// TIA Portal V21 export
FUNCTION_BLOCK "PHT Block"   // FB401, LAD
{ S7_Optimized_Access := 'FALSE' }
// stored: AutoNumber false, SetENOAutomatically false
   VAR_INPUT
      Secs : Bool;
      Start : Bool;
      Stop : Bool;
      Abort : Bool;
      AlarmAck : Bool;
      AlwaysTrue : Bool;
      StartupMsgSelection : Bool;
      spare1 : Bool;
      spare2 : Bool;
      EndMsgSelection : Bool;
      EndMsgAck : Bool;
      Fault : Bool;
      Popup1Enable : Bool;
      Popup2Enable : Bool;
      ScadaHmi : Bool := 1;   // 0- scada, 1 - hmi
      StabilizeTime : Int;
      SetPressure : Real;
      ReleasePressure : Real;
      FailPressure : Real;
      AcceptableLeakage : Real;
      HoldTime : Int;
      UtilityValveDelay : Int;
      "Actual Minimum Pressure" : Real;
      "Actual Maximum Pressure" : Real;
      MaximumAttemptToFailedSelection : Int;
      MaximumNoAttemptToFailed : Int;
      PrintInterval : Int;
   END_VAR
   VAR_OUTPUT
      StartupMsg1 : Bool;
      CycleOver : Bool;
      LineValves : Bool;
      ControlValve : Bool;
      UtilityValve : Bool;
      StartupMsg : Bool;
      EndMsg : Bool;
      TestPassAlarm : Bool;
      TestFailAlarm : Bool;
      DrainValves : Bool;
      StartupMsg2 : Bool;
      StabilizeActualSecs : DInt;
      HoldActualMins : DInt;
      HoldActualSecs : DInt;
      Status : Int;
      StatusStr : String[60];
      UtilityValveActualDelay : Int;
      Event : Word;
   END_VAR
   VAR_IN_OUT
      Selected : Bool;
      CycleSelected : Bool;
      Running : Bool;
      VesselPressurised : Bool;
      DataLogCmd : Bool;
      StartLog : Bool;
      EndLog : Bool;
      DataLogYes : Bool;
      ResetPhtTimer : Bool;
      VesselStabilised : Bool;
      DelayToConfirmVesselPressurized : Bool;
      PressureDropDuringStabilizeTime : Bool;
      PressureDropDuringHoldTime : Bool;
      TestPassedRW : Bool;
      DelayToStartReleaseDone : Bool;
      DrainValve : Bool;
      StabilizePopup : Bool;
      LineValvesOpeningTime : Int;
      DrainValvesOpeningTime : Int;
      AcceptablePressure : Real;
      "PHT Selected" : Bool;
      TestAborted : Bool;
      ResetBit : Bool;
      Popup2Ack : Bool;
      StartupMsgYes : Bool;
      StartupMsgNo : Bool;
      MaximumNoAttemptToFailedTemp : Int;
   END_VAR
   VAR
      StabilizeTimer { S7_SetPoint := 'True'} : "R_TIMER";
      HoldTimer { S7_SetPoint := 'True'} : "R_TIMER";
      CheckPressureDuringStabilizeTime { S7_SetPoint := 'True'} : "On Delay Timer";
      CheckPressureDuringHoldTime { S7_SetPoint := 'True'} : "On Delay Timer";
      ReleaseCheckTime { S7_SetPoint := 'True'} : "On Delay Timer";
      CheckPressuredelay { S7_SetPoint := 'True'} : "On Delay Timer";
      DelayToStartRelease { S7_SetPoint := 'True'} : "On Delay Timer";
      StabilizeDelay { S7_SetPoint := 'True'} : "On Delay Timer";
      IEC_Timer_0_Instance { S7_SetPoint := 'True'} : TON_TIME;
      IEC_Timer_1_Instance { S7_SetPoint := 'True'} : TON_TIME;
      Timer1 { S7_SetPoint := 'True'} : TON_TIME;
      Timer2 { S7_SetPoint := 'True'} : TON_TIME;
      Timer3 { S7_SetPoint := 'True'} : TON_TIME;
      Timer4 { S7_SetPoint := 'True'} : TON_TIME;
      Timer5 { S7_SetPoint := 'True'} : TON_TIME;
      Timer6 { S7_SetPoint := 'True'} : TON_TIME;
      Timer7 { S7_SetPoint := 'True'} : TON_TIME;
      Re { ExternalAccessible := 'False'; ExternalVisible := 'False'; ExternalWritable := 'False'} : Bool;
      Re1 { ExternalAccessible := 'False'; ExternalVisible := 'False'; ExternalWritable := 'False'} : Bool;
      Re2 { ExternalAccessible := 'False'; ExternalVisible := 'False'; ExternalWritable := 'False'} : Bool;
      Re3 { ExternalAccessible := 'False'; ExternalVisible := 'False'; ExternalWritable := 'False'} : Bool;
      Re4 { ExternalAccessible := 'False'; ExternalVisible := 'False'; ExternalWritable := 'False'} : Bool;
      Re5 { ExternalAccessible := 'False'; ExternalVisible := 'False'; ExternalWritable := 'False'} : Bool;
      Re6 { ExternalAccessible := 'False'; ExternalVisible := 'False'; ExternalWritable := 'False'} : Bool;
      Re7 { ExternalAccessible := 'False'; ExternalVisible := 'False'; ExternalWritable := 'False'} : Bool;
      Re8 { ExternalAccessible := 'False'; ExternalVisible := 'False'; ExternalWritable := 'False'} : Bool;
      Re9 { ExternalAccessible := 'False'; ExternalVisible := 'False'; ExternalWritable := 'False'} : Bool;
      Re10 : Bool;
      Re11 : Bool;
      Re12 : Bool;
      Timer8 : TON_TIME;
      Timer9 { S7_SetPoint := 'True'} : TON_TIME;
      Timer10 { S7_SetPoint := 'True'} : TON_TIME;
      Timer11 { S7_SetPoint := 'True'} : TON_TIME;
      Timer12 { S7_SetPoint := 'True'} : TON_TIME;
      IEC_Counter_0_Instance { S7_SetPoint := 'True'} : CTU_INT;
      Re13 : Bool;
      Re14 : Bool;
      Re15 : Bool;
      timer13 : TON_TIME;
   END_VAR
   VAR_TEMP   // added for the SCL form of the ladder/FBD networks
      _w1 : Bool;
      _w2 : Bool;
      _w3 : Bool;
      _w4 : Bool;
      _w5 : Bool;
      _w6 : Bool;
      _w7 : Bool;
      _w8 : Bool;
      _w9 : Bool;
      _w10 : Bool;
      _w11 : Bool;
      _w12 : Bool;
      _w13 : Bool;
      _w14 : Bool;
      _w15 : Bool;
      _w16 : Bool;
   END_VAR
BEGIN

REGION Network 1: StartupMsgYesEnable
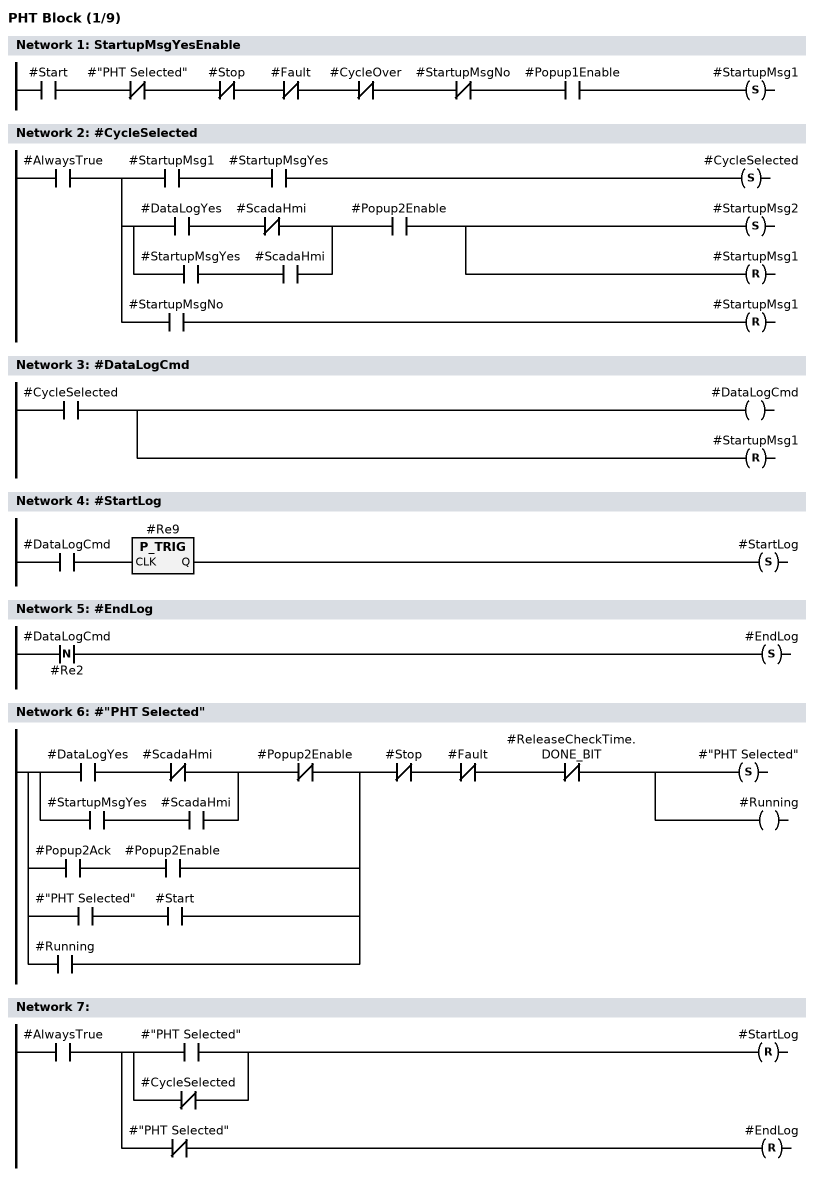
   RUNG wire#powerrail
      Contact( #Start )
      I_Contact( #"PHT Selected" )
      I_Contact( #Stop )
      I_Contact( #Fault )
      I_Contact( #CycleOver )
      I_Contact( #StartupMsgNo )
      Contact( #Popup1Enable )
      S_Coil( #StartupMsg1 )
   END_RUNG
   // the same network as SCL:
   IF #Start AND NOT #"PHT Selected" AND NOT #Stop AND NOT #Fault AND NOT #CycleOver AND NOT #StartupMsgNo AND #Popup1Enable THEN
       #StartupMsg1 := TRUE;
   END_IF;
END_REGION

REGION Network 2: #CycleSelected
   RUNG wire#powerrail
      Contact( #AlwaysTrue )
      wire#w1
      Contact( #StartupMsg1 )
      Contact( #StartupMsgYes )
      S_Coil( #CycleSelected )
   END_RUNG
   RUNG wire#w1
      Contact( #DataLogYes )
      I_Contact( #ScadaHmi )
      wire#w2
      Contact( #Popup2Enable )
      wire#w3
      S_Coil( #StartupMsg2 )
   END_RUNG
   RUNG wire#w1
      Contact( #StartupMsgYes )
      Contact( #ScadaHmi )
   END_RUNG wire#w2
   RUNG wire#w3
      R_Coil( #StartupMsg1 )
   END_RUNG
   RUNG wire#w1
      Contact( #StartupMsgNo )
      R_Coil( #StartupMsg1 )
   END_RUNG
   // the same network as SCL:
   IF #AlwaysTrue AND #StartupMsg1 AND #StartupMsgYes THEN #CycleSelected := TRUE; END_IF;
   IF #AlwaysTrue AND ((#DataLogYes AND NOT #ScadaHmi) OR (#StartupMsgYes AND #ScadaHmi)) AND #Popup2Enable THEN
       #StartupMsg2 := TRUE;
       #StartupMsg1 := FALSE;
   END_IF;
   IF #AlwaysTrue AND #StartupMsgNo THEN #StartupMsg1 := FALSE; END_IF;
END_REGION

REGION Network 3: #DataLogCmd
   RUNG wire#powerrail
      Contact( #CycleSelected )
      wire#w1
      Coil( #DataLogCmd )
   END_RUNG
   RUNG wire#w1
      R_Coil( #StartupMsg1 )
   END_RUNG
   // the same network as SCL:
   #DataLogCmd := #CycleSelected;
   IF #CycleSelected THEN #StartupMsg1 := FALSE; END_IF;
END_REGION

REGION Network 4: #StartLog
   RUNG wire#powerrail
      Contact( #DataLogCmd )
      P_Trig( #Re9 )
      S_Coil( #StartLog )
   END_RUNG
   // the same network as SCL:
   #_w1 := #DataLogCmd AND NOT #Re9;   // rising edge
   #Re9 := #DataLogCmd;
   IF #_w1 THEN #StartLog := TRUE; END_IF;
END_REGION

REGION Network 5: #EndLog
   RUNG wire#powerrail
      N_Contact(operand := #DataLogCmd, bit := #Re2)
      S_Coil( #EndLog )
   END_RUNG
   // the same network as SCL:
   #_w1 := NOT #DataLogCmd AND #Re2;   // falling edge of #DataLogCmd
   #Re2 := #DataLogCmd;
   IF #_w1 THEN #EndLog := TRUE; END_IF;
END_REGION

REGION Network 6: #"PHT Selected"
   RUNG wire#powerrail
      Contact( #DataLogYes )
      I_Contact( #ScadaHmi )
      wire#w1
      I_Contact( #Popup2Enable )
      wire#w2
      I_Contact( #Stop )
      I_Contact( #Fault )
      I_Contact( #ReleaseCheckTime.DONE_BIT )
      wire#w3
      S_Coil( #"PHT Selected" )
   END_RUNG
   RUNG wire#powerrail
      Contact( #StartupMsgYes )
      Contact( #ScadaHmi )
   END_RUNG wire#w1
   RUNG wire#powerrail
      Contact( #Popup2Ack )
      Contact( #Popup2Enable )
   END_RUNG wire#w2
   RUNG wire#powerrail
      Contact( #"PHT Selected" )
      Contact( #Start )
   END_RUNG wire#w2
   RUNG wire#powerrail
      Contact( #Running )
   END_RUNG wire#w2
   RUNG wire#w3
      Coil( #Running )
   END_RUNG
   // the same network as SCL:
   #_w1 := ((((#DataLogYes AND NOT #ScadaHmi) OR (#StartupMsgYes AND #ScadaHmi)) AND NOT #Popup2Enable) OR (#Popup2Ack AND #Popup2Enable) OR (#"PHT Selected" AND #Start) OR #Running) AND NOT #Stop AND NOT #Fault AND NOT #ReleaseCheckTime.DONE_BIT;
   IF #_w1 THEN #"PHT Selected" := TRUE; END_IF;
   #Running := #_w1;
END_REGION

REGION Network 7
   RUNG wire#powerrail
      Contact( #AlwaysTrue )
      wire#w1
      Contact( #"PHT Selected" )
      wire#w2
      R_Coil( #StartLog )
   END_RUNG
   RUNG wire#w1
      I_Contact( #CycleSelected )
   END_RUNG wire#w2
   RUNG wire#w1
      I_Contact( #"PHT Selected" )
      R_Coil( #EndLog )
   END_RUNG
   // the same network as SCL:
   IF #AlwaysTrue AND (#"PHT Selected" OR NOT #CycleSelected) THEN #StartLog := FALSE; END_IF;
   IF #AlwaysTrue AND NOT #"PHT Selected" THEN #EndLog := FALSE; END_IF;
END_REGION

REGION Network 8: OUTPUT ON
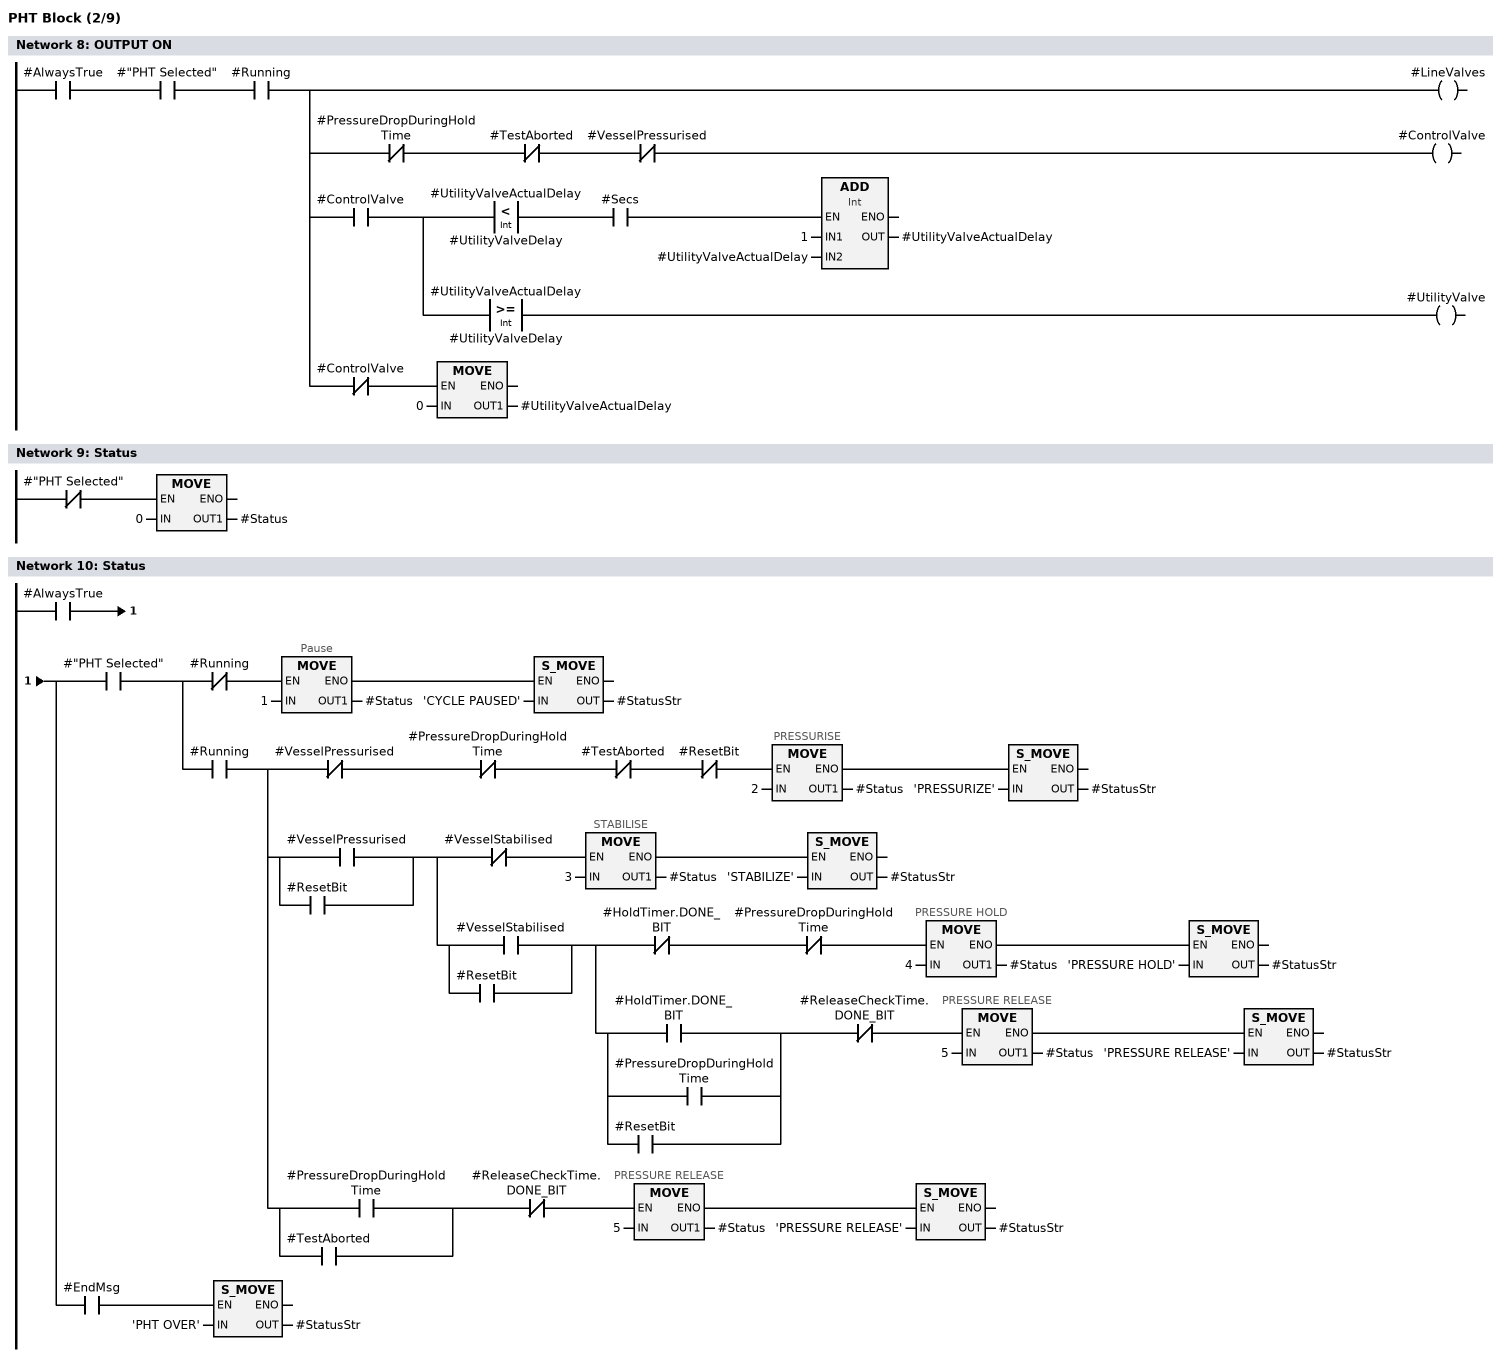
   RUNG wire#powerrail
      Contact( #AlwaysTrue )
      Contact( #"PHT Selected" )
      Contact( #Running )
      wire#w1
      Coil( #LineValves )
   END_RUNG
   RUNG wire#w1
      I_Contact( #PressureDropDuringHoldTime )
      I_Contact( #TestAborted )
      I_Contact( #VesselPressurised )
      Coil( #ControlValve )
   END_RUNG
   RUNG wire#w1
      Contact( #ControlValve )
      wire#w2
      { S7_Templates := "SrcType := Int" } LT_Contact(in1 := #UtilityValveActualDelay, in2 := #UtilityValveDelay)
      Contact( #Secs )
      { S7_Templates := "SrcType := Int" } Add(in1 := 1, in2 := #UtilityValveActualDelay, out => #UtilityValveActualDelay)
   END_RUNG
   RUNG wire#w2
      { S7_Templates := "SrcType := Int" } GE_Contact(in1 := #UtilityValveActualDelay, in2 := #UtilityValveDelay)
      Coil( #UtilityValve )
   END_RUNG
   RUNG wire#w1
      I_Contact( #ControlValve )
      Move(in := 0, out1 => #UtilityValveActualDelay)
   END_RUNG
   // the same network as SCL:
   #LineValves := #AlwaysTrue AND #"PHT Selected" AND #Running;
   #ControlValve := #LineValves AND NOT #PressureDropDuringHoldTime AND NOT #TestAborted AND NOT #VesselPressurised;
   #_w1 := #LineValves AND #ControlValve;
   IF #_w1 AND (#UtilityValveActualDelay < #UtilityValveDelay) AND #Secs THEN
       #UtilityValveActualDelay := 1 + #UtilityValveActualDelay;
   END_IF;
   #UtilityValve := #_w1 AND (#UtilityValveActualDelay >= #UtilityValveDelay);
   IF #LineValves AND NOT #ControlValve THEN #UtilityValveActualDelay := 0; END_IF;
END_REGION

REGION Network 9: Status
   RUNG wire#powerrail
      I_Contact( #"PHT Selected" )
      { S7_GenerateENO := "TRUE" } Move(in := 0, out1 => #Status)
   END_RUNG
   // the same network as SCL:
   IF NOT #"PHT Selected" THEN #Status := 0; END_IF;
END_REGION

REGION Network 10: Status
   RUNG wire#powerrail
      Contact( #AlwaysTrue )
      wire#w1
      Contact( #"PHT Selected" )
      wire#w2
      I_Contact( #Running )
      { S7_GenerateENO := "TRUE" } Move(in := 1, out1 => #Status)   // Pause
      S_Move(in := 'CYCLE PAUSED', out => #StatusStr)
   END_RUNG
   RUNG wire#w2
      Contact( #Running )
      wire#w3
      I_Contact( #VesselPressurised )
      I_Contact( #PressureDropDuringHoldTime )
      I_Contact( #TestAborted )
      I_Contact( #ResetBit )
      { S7_GenerateENO := "TRUE" } Move(in := 2, out1 => #Status)   // PRESSURISE
      S_Move(in := 'PRESSURIZE', out => #StatusStr)
   END_RUNG
   RUNG wire#w3
      Contact( #VesselPressurised )
      wire#w4
      I_Contact( #VesselStabilised )
      { S7_GenerateENO := "TRUE" } Move(in := 3, out1 => #Status)   // STABILISE
      S_Move(in := 'STABILIZE', out => #StatusStr)
   END_RUNG
   RUNG wire#w3
      Contact( #ResetBit )
   END_RUNG wire#w4
   RUNG wire#w4
      Contact( #VesselStabilised )
      wire#w5
      I_Contact( #HoldTimer.DONE_BIT )
      I_Contact( #PressureDropDuringHoldTime )
      { S7_GenerateENO := "TRUE" } Move(in := 4, out1 => #Status)   // PRESSURE HOLD
      S_Move(in := 'PRESSURE HOLD', out => #StatusStr)
   END_RUNG
   RUNG wire#w4
      Contact( #ResetBit )
   END_RUNG wire#w5
   RUNG wire#w5
      Contact( #HoldTimer.DONE_BIT )
      wire#w6
      I_Contact( #ReleaseCheckTime.DONE_BIT )
      { S7_GenerateENO := "TRUE" } Move(in := 5, out1 => #Status)   // PRESSURE RELEASE
      S_Move(in := 'PRESSURE RELEASE', out => #StatusStr)
   END_RUNG
   RUNG wire#w5
      Contact( #PressureDropDuringHoldTime )
   END_RUNG wire#w6
   RUNG wire#w5
      Contact( #ResetBit )
   END_RUNG wire#w6
   RUNG wire#w3
      Contact( #PressureDropDuringHoldTime )
      wire#w7
      I_Contact( #ReleaseCheckTime.DONE_BIT )
      { S7_GenerateENO := "TRUE" } Move(in := 5, out1 => #Status)   // PRESSURE RELEASE
      S_Move(in := 'PRESSURE RELEASE', out => #StatusStr)
   END_RUNG
   RUNG wire#w3
      Contact( #TestAborted )
   END_RUNG wire#w7
   RUNG wire#w1
      Contact( #EndMsg )
      S_Move(in := 'PHT OVER', out => #StatusStr)
   END_RUNG
   // the same network as SCL:
   // ENO of a box is taken as its EN; it also drops when the box reports an error
   #_w1 := #AlwaysTrue AND #"PHT Selected";
   IF #_w1 AND NOT #Running THEN
       #Status := 1;   // Pause
       #StatusStr := 'CYCLE PAUSED';
   END_IF;
   #_w2 := #_w1 AND #Running;
   IF #_w2 AND NOT #VesselPressurised AND NOT #PressureDropDuringHoldTime AND NOT #TestAborted AND NOT #ResetBit THEN
       #Status := 2;   // PRESSURISE
       #StatusStr := 'PRESSURIZE';
   END_IF;
   #_w3 := #_w2 AND (#VesselPressurised OR #ResetBit);
   IF #_w3 AND NOT #VesselStabilised THEN
       #Status := 3;   // STABILISE
       #StatusStr := 'STABILIZE';
   END_IF;
   #_w4 := #_w3 AND (#VesselStabilised OR #ResetBit);
   IF #_w4 AND NOT #HoldTimer.DONE_BIT AND NOT #PressureDropDuringHoldTime THEN
       #Status := 4;   // PRESSURE HOLD
       #StatusStr := 'PRESSURE HOLD';
   END_IF;
   IF #_w4 AND (#HoldTimer.DONE_BIT OR #PressureDropDuringHoldTime OR #ResetBit) AND NOT #ReleaseCheckTime.DONE_BIT THEN
       #Status := 5;   // PRESSURE RELEASE
       #StatusStr := 'PRESSURE RELEASE';
   END_IF;
   IF #_w2 AND (#PressureDropDuringHoldTime OR #TestAborted) AND NOT #ReleaseCheckTime.DONE_BIT THEN
       #Status := 5;   // PRESSURE RELEASE
       #StatusStr := 'PRESSURE RELEASE';
   END_IF;
   IF #AlwaysTrue AND #EndMsg THEN #StatusStr := 'PHT OVER'; END_IF;
END_REGION

REGION Network 11: Delays for opening drain valves
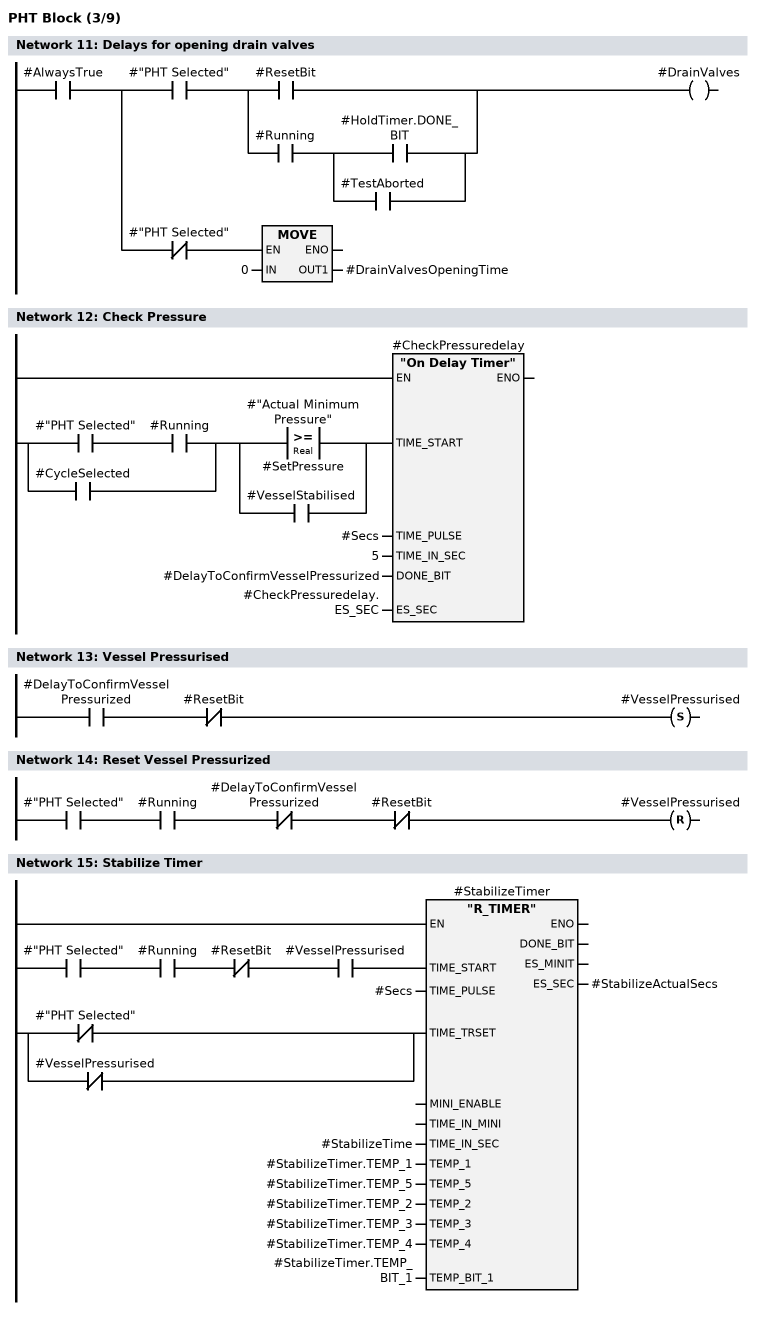
   RUNG wire#powerrail
      Contact( #AlwaysTrue )
      wire#w1
      Contact( #"PHT Selected" )
      wire#w2
      Contact( #ResetBit )
      wire#w3
      Coil( #DrainValves )
   END_RUNG
   RUNG wire#w2
      Contact( #Running )
      wire#w4
      Contact( #HoldTimer.DONE_BIT )
   END_RUNG wire#w3
   RUNG wire#w4
      Contact( #TestAborted )
   END_RUNG wire#w3
   RUNG wire#w1
      I_Contact( #"PHT Selected" )
      { S7_GenerateENO := "TRUE" } Move(in := 0, out1 => #DrainValvesOpeningTime)
   END_RUNG
   // the same network as SCL:
   #DrainValves := #AlwaysTrue AND #"PHT Selected" AND (#ResetBit OR (#Running AND (#HoldTimer.DONE_BIT OR #TestAborted)));
   IF #AlwaysTrue AND NOT #"PHT Selected" THEN #DrainValvesOpeningTime := 0; END_IF;
END_REGION

REGION Network 12: Check Pressure
   RUNG wire#powerrail
      #CheckPressuredelay(TIME_START := wire#w2, TIME_PULSE := #Secs, TIME_IN_SEC := 5, DONE_BIT := #DelayToConfirmVesselPressurized, ES_SEC := #CheckPressuredelay.ES_SEC)
   END_RUNG
   RUNG wire#powerrail
      Contact( #"PHT Selected" )
      Contact( #Running )
      wire#w1
      { S7_Templates := "SrcType := Real" } GE_Contact(in1 := #"Actual Minimum Pressure", in2 := #SetPressure)
   END_RUNG wire#w2
   RUNG wire#powerrail
      Contact( #CycleSelected )
   END_RUNG wire#w1
   RUNG wire#w1
      Contact( #VesselStabilised )
   END_RUNG wire#w2
   // the same network as SCL:
   #CheckPressuredelay(TIME_START := ((#"PHT Selected" AND #Running) OR #CycleSelected) AND ((#"Actual Minimum Pressure" >= #SetPressure) OR #VesselStabilised),   // "On Delay Timer"
                       TIME_PULSE := #Secs,
                       TIME_IN_SEC := 5,
                       DONE_BIT := #DelayToConfirmVesselPressurized,
                       ES_SEC := #CheckPressuredelay.ES_SEC);
END_REGION

REGION Network 13: Vessel Pressurised
   RUNG wire#powerrail
      Contact( #DelayToConfirmVesselPressurized )
      I_Contact( #ResetBit )
      S_Coil( #VesselPressurised )
   END_RUNG
   // the same network as SCL:
   IF #DelayToConfirmVesselPressurized AND NOT #ResetBit THEN #VesselPressurised := TRUE; END_IF;
END_REGION

REGION Network 14: Reset Vessel Pressurized
   RUNG wire#powerrail
      Contact( #"PHT Selected" )
      Contact( #Running )
      I_Contact( #DelayToConfirmVesselPressurized )
      I_Contact( #ResetBit )
      R_Coil( #VesselPressurised )
   END_RUNG
   // the same network as SCL:
   IF #"PHT Selected" AND #Running AND NOT #DelayToConfirmVesselPressurized AND NOT #ResetBit THEN
       #VesselPressurised := FALSE;
   END_IF;
END_REGION

REGION Network 15: Stabilize Timer
   RUNG wire#powerrail
      #StabilizeTimer(TIME_START := wire#w1, TIME_TRSET := wire#w2, TIME_PULSE := #Secs, MINI_ENABLE :=, TIME_IN_MINI :=, TIME_IN_SEC := #StabilizeTime, TEMP_1 := #StabilizeTimer.TEMP_1, TEMP_5 := #StabilizeTimer.TEMP_5, TEMP_2 := #StabilizeTimer.TEMP_2, TEMP_3 := #StabilizeTimer.TEMP_3, TEMP_4 := #StabilizeTimer.TEMP_4, TEMP_BIT_1 := #StabilizeTimer.TEMP_BIT_1, DONE_BIT =>, ES_MINIT =>, ES_SEC => #StabilizeActualSecs)
   END_RUNG
   RUNG wire#powerrail
      Contact( #"PHT Selected" )
      Contact( #Running )
      I_Contact( #ResetBit )
      Contact( #VesselPressurised )
   END_RUNG wire#w1
   RUNG wire#powerrail
      I_Contact( #"PHT Selected" )
   END_RUNG wire#w2
   RUNG wire#powerrail
      I_Contact( #VesselPressurised )
   END_RUNG wire#w2
   // the same network as SCL:
   #StabilizeTimer(TIME_START := #"PHT Selected" AND #Running AND NOT #ResetBit AND #VesselPressurised,   // "R_TIMER"
                   TIME_PULSE := #Secs,
                   TIME_TRSET := NOT #"PHT Selected" OR NOT #VesselPressurised,
                   TIME_IN_SEC := #StabilizeTime,
                   TEMP_1 := #StabilizeTimer.TEMP_1,
                   TEMP_5 := #StabilizeTimer.TEMP_5,
                   TEMP_2 := #StabilizeTimer.TEMP_2,
                   TEMP_3 := #StabilizeTimer.TEMP_3,
                   TEMP_4 := #StabilizeTimer.TEMP_4,
                   TEMP_BIT_1 := #StabilizeTimer.TEMP_BIT_1,
                   ES_SEC => #StabilizeActualSecs);
END_REGION

REGION Network 16: Check Pressure During Stabilize
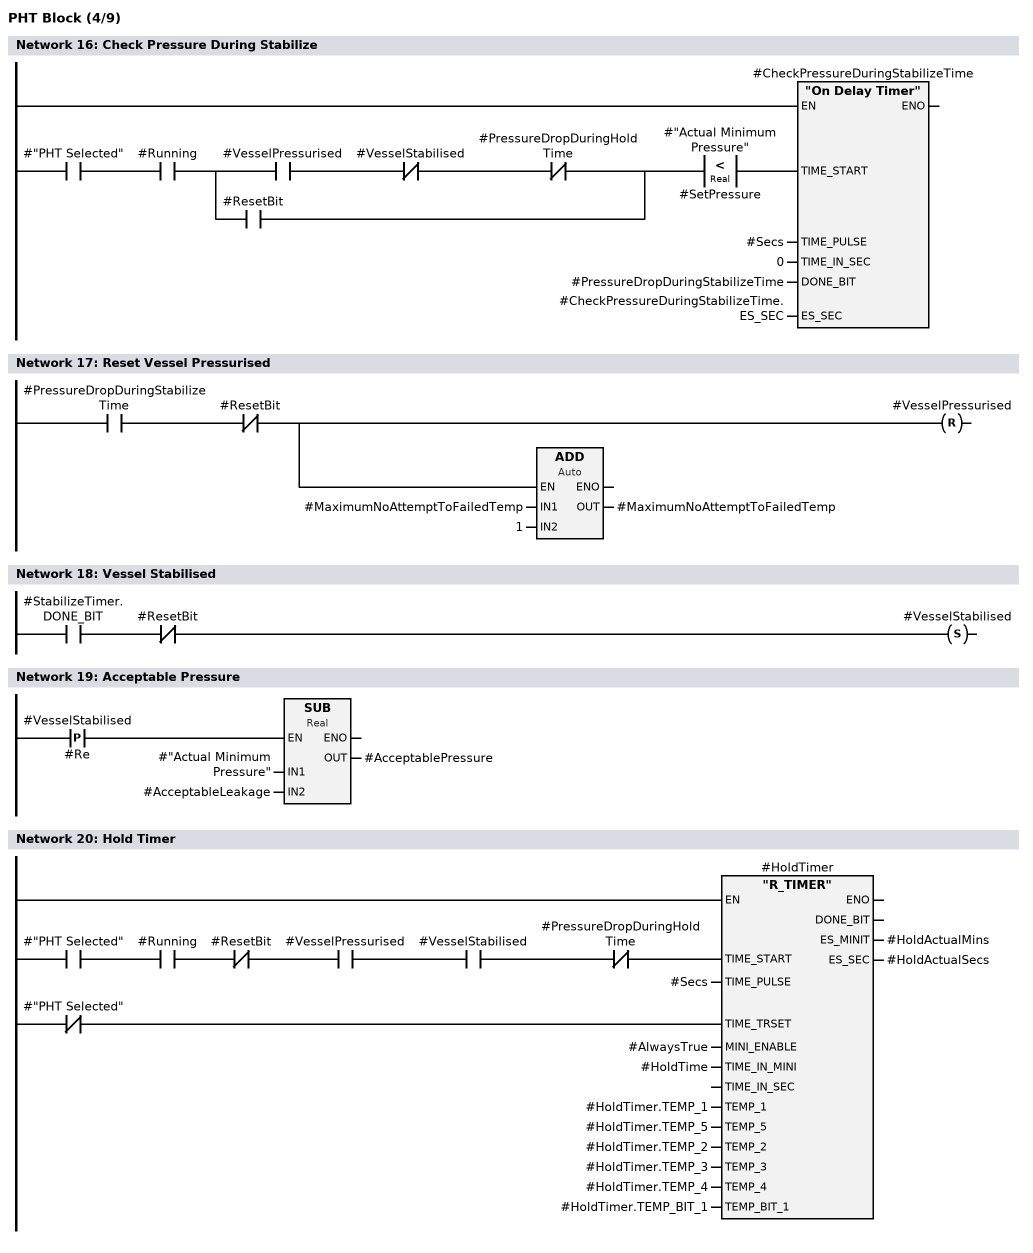
   RUNG wire#powerrail
      #CheckPressureDuringStabilizeTime(TIME_START := wire#w3, TIME_PULSE := #Secs, TIME_IN_SEC := 0, DONE_BIT := #PressureDropDuringStabilizeTime, ES_SEC := #CheckPressureDuringStabilizeTime.ES_SEC)
   END_RUNG
   RUNG wire#powerrail
      Contact( #"PHT Selected" )
      Contact( #Running )
      wire#w1
      Contact( #VesselPressurised )
      I_Contact( #VesselStabilised )
      I_Contact( #PressureDropDuringHoldTime )
      wire#w2
      { S7_Templates := "SrcType := Real" } LT_Contact(in1 := #"Actual Minimum Pressure", in2 := #SetPressure)
   END_RUNG wire#w3
   RUNG wire#w1
      Contact( #ResetBit )
   END_RUNG wire#w2
   // the same network as SCL:
   #CheckPressureDuringStabilizeTime(TIME_START := #"PHT Selected" AND #Running AND ((#VesselPressurised AND NOT #VesselStabilised AND NOT #PressureDropDuringHoldTime) OR #ResetBit) AND (#"Actual Minimum Pressure" < #SetPressure),   // "On Delay Timer"
                           TIME_PULSE := #Secs,
                           TIME_IN_SEC := 0,
                           DONE_BIT := #PressureDropDuringStabilizeTime,
                           ES_SEC := #CheckPressureDuringStabilizeTime.ES_SEC);
END_REGION

REGION Network 17: Reset Vessel Pressurised
   RUNG wire#powerrail
      Contact( #PressureDropDuringStabilizeTime )
      I_Contact( #ResetBit )
      wire#w1
      R_Coil( #VesselPressurised )
   END_RUNG
   RUNG wire#w1
      Add(in1 := #MaximumNoAttemptToFailedTemp, in2 := 1, out => #MaximumNoAttemptToFailedTemp)
   END_RUNG
   // the same network as SCL:
   IF #PressureDropDuringStabilizeTime AND NOT #ResetBit THEN
       #VesselPressurised := FALSE;
       #MaximumNoAttemptToFailedTemp := #MaximumNoAttemptToFailedTemp + 1;
   END_IF;
END_REGION

REGION Network 18: Vessel Stabilised
   RUNG wire#powerrail
      Contact( #StabilizeTimer.DONE_BIT )
      I_Contact( #ResetBit )
      S_Coil( #VesselStabilised )
   END_RUNG
   // the same network as SCL:
   IF #StabilizeTimer.DONE_BIT AND NOT #ResetBit THEN #VesselStabilised := TRUE; END_IF;
END_REGION

REGION Network 19: Acceptable Pressure
   RUNG wire#powerrail
      P_Contact(operand := #VesselStabilised, bit := #Re)
      { S7_Templates := "SrcType := Real"; S7_GenerateENO := "TRUE" } Sub(in1 := #"Actual Minimum Pressure", in2 := #AcceptableLeakage, out => #AcceptablePressure)
   END_RUNG
   // the same network as SCL:
   #_w1 := #VesselStabilised AND NOT #Re;   // rising edge of #VesselStabilised
   #Re := #VesselStabilised;
   IF #_w1 THEN #AcceptablePressure := #"Actual Minimum Pressure" - #AcceptableLeakage; END_IF;
END_REGION

REGION Network 20: Hold Timer
   RUNG wire#powerrail
      #HoldTimer(TIME_START := wire#w1, TIME_TRSET := wire#w2, TIME_PULSE := #Secs, MINI_ENABLE := #AlwaysTrue, TIME_IN_MINI := #HoldTime, TIME_IN_SEC :=, TEMP_1 := #HoldTimer.TEMP_1, TEMP_5 := #HoldTimer.TEMP_5, TEMP_2 := #HoldTimer.TEMP_2, TEMP_3 := #HoldTimer.TEMP_3, TEMP_4 := #HoldTimer.TEMP_4, TEMP_BIT_1 := #HoldTimer.TEMP_BIT_1, DONE_BIT =>, ES_MINIT => #HoldActualMins, ES_SEC => #HoldActualSecs)
   END_RUNG
   RUNG wire#powerrail
      Contact( #"PHT Selected" )
      Contact( #Running )
      I_Contact( #ResetBit )
      Contact( #VesselPressurised )
      Contact( #VesselStabilised )
      I_Contact( #PressureDropDuringHoldTime )
   END_RUNG wire#w1
   RUNG wire#powerrail
      I_Contact( #"PHT Selected" )
   END_RUNG wire#w2
   // the same network as SCL:
   #HoldTimer(TIME_START := #"PHT Selected" AND #Running AND NOT #ResetBit AND #VesselPressurised AND #VesselStabilised AND NOT #PressureDropDuringHoldTime,   // "R_TIMER"
              TIME_PULSE := #Secs,
              TIME_TRSET := NOT #"PHT Selected",
              MINI_ENABLE := #AlwaysTrue,
              TIME_IN_MINI := #HoldTime,
              TEMP_1 := #HoldTimer.TEMP_1,
              TEMP_5 := #HoldTimer.TEMP_5,
              TEMP_2 := #HoldTimer.TEMP_2,
              TEMP_3 := #HoldTimer.TEMP_3,
              TEMP_4 := #HoldTimer.TEMP_4,
              TEMP_BIT_1 := #HoldTimer.TEMP_BIT_1,
              ES_MINIT => #HoldActualMins,
              ES_SEC => #HoldActualSecs);
END_REGION

REGION Network 21: Check Pressure to abort Cycle during Hold Time
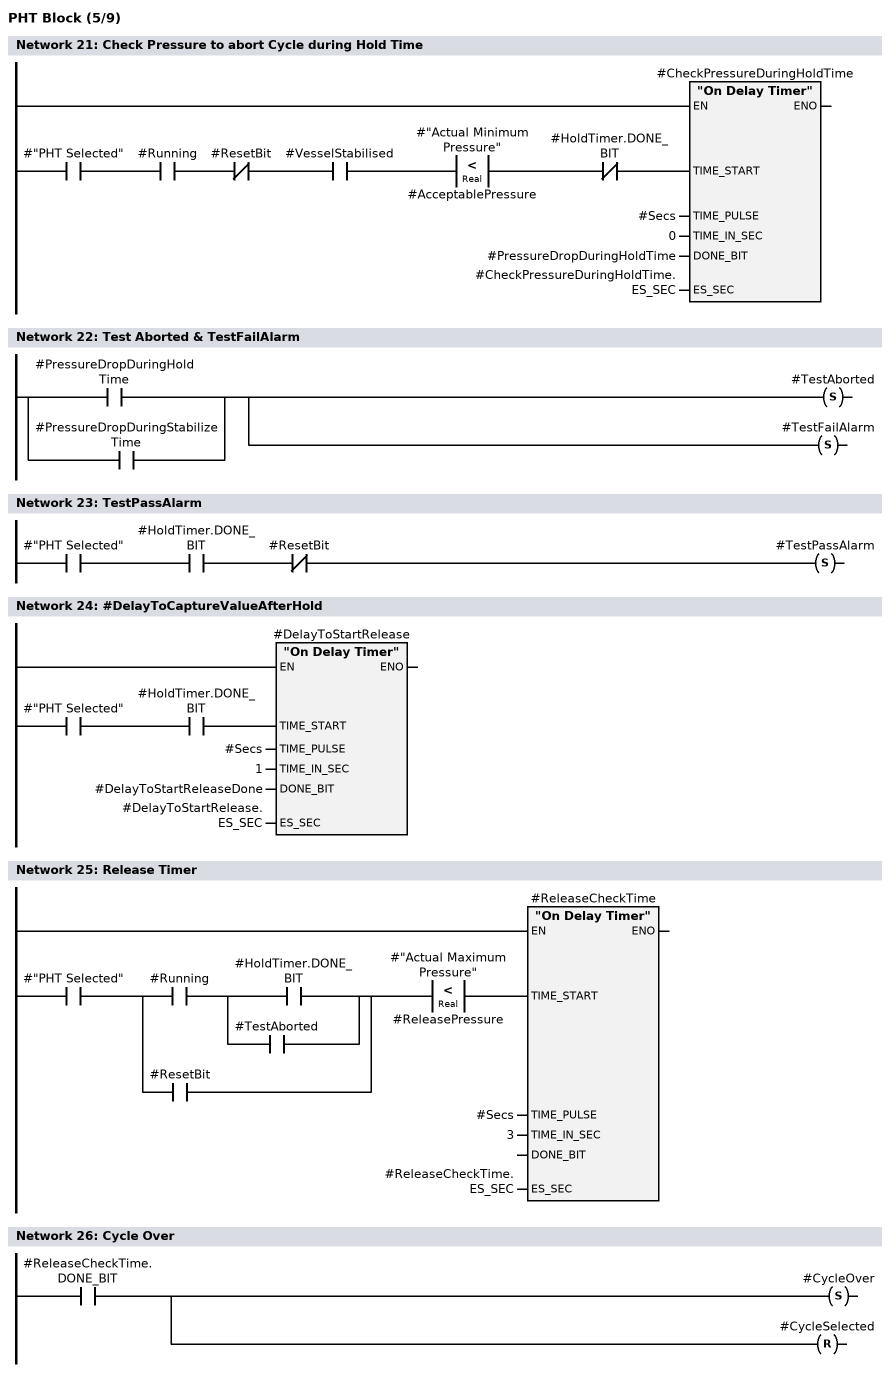
   RUNG wire#powerrail
      #CheckPressureDuringHoldTime(TIME_START := wire#w1, TIME_PULSE := #Secs, TIME_IN_SEC := 0, DONE_BIT := #PressureDropDuringHoldTime, ES_SEC := #CheckPressureDuringHoldTime.ES_SEC)
   END_RUNG
   RUNG wire#powerrail
      Contact( #"PHT Selected" )
      Contact( #Running )
      I_Contact( #ResetBit )
      Contact( #VesselStabilised )
      { S7_Templates := "SrcType := Real" } LT_Contact(in1 := #"Actual Minimum Pressure", in2 := #AcceptablePressure)
      I_Contact( #HoldTimer.DONE_BIT )
   END_RUNG wire#w1
   // the same network as SCL:
   #CheckPressureDuringHoldTime(TIME_START := #"PHT Selected" AND #Running AND NOT #ResetBit AND #VesselStabilised AND (#"Actual Minimum Pressure" < #AcceptablePressure) AND NOT #HoldTimer.DONE_BIT,   // "On Delay Timer"
                           TIME_PULSE := #Secs,
                           TIME_IN_SEC := 0,
                           DONE_BIT := #PressureDropDuringHoldTime,
                           ES_SEC := #CheckPressureDuringHoldTime.ES_SEC);
END_REGION

REGION Network 22: Test Aborted & TestFailAlarm
   RUNG wire#powerrail
      Contact( #PressureDropDuringHoldTime )
      wire#w1
      S_Coil( #TestAborted )
   END_RUNG
   RUNG wire#powerrail
      Contact( #PressureDropDuringStabilizeTime )
   END_RUNG wire#w1
   RUNG wire#w1
      S_Coil( #TestFailAlarm )
   END_RUNG
   // the same network as SCL:
   IF #PressureDropDuringHoldTime OR #PressureDropDuringStabilizeTime THEN
       #TestAborted := TRUE;
       #TestFailAlarm := TRUE;
   END_IF;
END_REGION

REGION Network 23: TestPassAlarm
   RUNG wire#powerrail
      Contact( #"PHT Selected" )
      Contact( #HoldTimer.DONE_BIT )
      I_Contact( #ResetBit )
      S_Coil( #TestPassAlarm )
   END_RUNG
   // the same network as SCL:
   IF #"PHT Selected" AND #HoldTimer.DONE_BIT AND NOT #ResetBit THEN #TestPassAlarm := TRUE; END_IF;
END_REGION

REGION Network 24: #DelayToCaptureValueAfterHold
   RUNG wire#powerrail
      #DelayToStartRelease(TIME_START := wire#w1, TIME_PULSE := #Secs, TIME_IN_SEC := 1, DONE_BIT := #DelayToStartReleaseDone, ES_SEC := #DelayToStartRelease.ES_SEC)
   END_RUNG
   RUNG wire#powerrail
      Contact( #"PHT Selected" )
      Contact( #HoldTimer.DONE_BIT )
   END_RUNG wire#w1
   // the same network as SCL:
   #DelayToStartRelease(TIME_START := #"PHT Selected" AND #HoldTimer.DONE_BIT,   // "On Delay Timer"
                        TIME_PULSE := #Secs,
                        TIME_IN_SEC := 1,
                        DONE_BIT := #DelayToStartReleaseDone,
                        ES_SEC := #DelayToStartRelease.ES_SEC);
END_REGION

REGION Network 25: Release Timer
   RUNG wire#powerrail
      #ReleaseCheckTime(TIME_START := wire#w4, TIME_PULSE := #Secs, TIME_IN_SEC := 3, DONE_BIT :=, ES_SEC := #ReleaseCheckTime.ES_SEC)
   END_RUNG
   RUNG wire#powerrail
      Contact( #"PHT Selected" )
      wire#w1
      Contact( #Running )
      wire#w2
      Contact( #HoldTimer.DONE_BIT )
      wire#w3
      { S7_Templates := "SrcType := Real" } LT_Contact(in1 := #"Actual Maximum Pressure", in2 := #ReleasePressure)
   END_RUNG wire#w4
   RUNG wire#w2
      Contact( #TestAborted )
   END_RUNG wire#w3
   RUNG wire#w1
      Contact( #ResetBit )
   END_RUNG wire#w3
   // the same network as SCL:
   #ReleaseCheckTime(TIME_START := #"PHT Selected" AND ((#Running AND (#HoldTimer.DONE_BIT OR #TestAborted)) OR #ResetBit) AND (#"Actual Maximum Pressure" < #ReleasePressure),   // "On Delay Timer"
                     TIME_PULSE := #Secs,
                     TIME_IN_SEC := 3,
                     ES_SEC := #ReleaseCheckTime.ES_SEC);
END_REGION

REGION Network 26: Cycle Over
   RUNG wire#powerrail
      Contact( #ReleaseCheckTime.DONE_BIT )
      wire#w1
      S_Coil( #CycleOver )
   END_RUNG
   RUNG wire#w1
      R_Coil( #CycleSelected )
   END_RUNG
   // the same network as SCL:
   IF #ReleaseCheckTime.DONE_BIT THEN
       #CycleOver := TRUE;
       #CycleSelected := FALSE;
   END_IF;
END_REGION

REGION Network 27: Alarm Ack
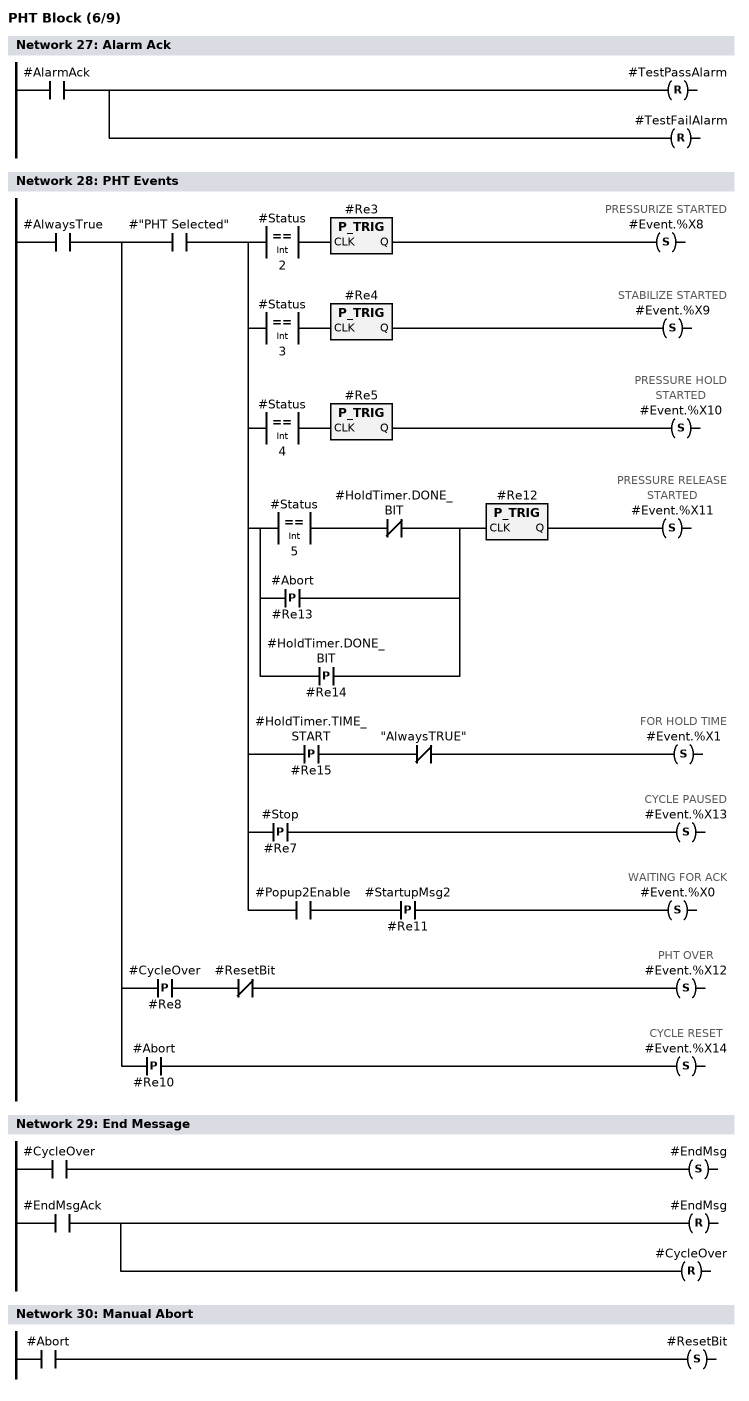
   RUNG wire#powerrail
      Contact( #AlarmAck )
      wire#w1
      R_Coil( #TestPassAlarm )
   END_RUNG
   RUNG wire#w1
      R_Coil( #TestFailAlarm )
   END_RUNG
   // the same network as SCL:
   IF #AlarmAck THEN
       #TestPassAlarm := FALSE;
       #TestFailAlarm := FALSE;
   END_IF;
END_REGION

REGION Network 28: PHT Events
   RUNG wire#powerrail
      Contact( #AlwaysTrue )
      wire#w1
      Contact( #"PHT Selected" )
      wire#w2
      { S7_Templates := "SrcType := Int" } EQ_Contact(in1 := #Status, in2 := 2)
      P_Trig( #Re3 )
      S_Coil( #Event.%X8 )   // PRESSURIZE STARTED
   END_RUNG
   RUNG wire#w2
      { S7_Templates := "SrcType := Int" } EQ_Contact(in1 := #Status, in2 := 3)
      P_Trig( #Re4 )
      S_Coil( #Event.%X9 )   // STABILIZE STARTED
   END_RUNG
   RUNG wire#w2
      { S7_Templates := "SrcType := Int" } EQ_Contact(in1 := #Status, in2 := 4)
      P_Trig( #Re5 )
      S_Coil( #Event.%X10 )   // PRESSURE HOLD STARTED
   END_RUNG
   RUNG wire#w2
      { S7_Templates := "SrcType := Int" } EQ_Contact(in1 := #Status, in2 := 5)
      I_Contact( #HoldTimer.DONE_BIT )
      wire#w3
      P_Trig( #Re12 )
      S_Coil( #Event.%X11 )   // PRESSURE RELEASE STARTED
   END_RUNG
   RUNG wire#w2
      P_Contact(operand := #Abort, bit := #Re13)
   END_RUNG wire#w3
   RUNG wire#w2
      P_Contact(operand := #HoldTimer.DONE_BIT, bit := #Re14)
   END_RUNG wire#w3
   RUNG wire#w2
      P_Contact(operand := #HoldTimer.TIME_START, bit := #Re15)
      I_Contact( "AlwaysTRUE" )
      S_Coil( #Event.%X1 )   // FOR HOLD TIME
   END_RUNG
   RUNG wire#w2
      P_Contact(operand := #Stop, bit := #Re7)
      S_Coil( #Event.%X13 )   // CYCLE PAUSED
   END_RUNG
   RUNG wire#w2
      Contact( #Popup2Enable )
      P_Contact(operand := #StartupMsg2, bit := #Re11)
      S_Coil( #Event.%X0 )   // WAITING FOR ACK
   END_RUNG
   RUNG wire#w1
      P_Contact(operand := #CycleOver, bit := #Re8)
      I_Contact( #ResetBit )
      S_Coil( #Event.%X12 )   // PHT OVER
   END_RUNG
   RUNG wire#w1
      P_Contact(operand := #Abort, bit := #Re10)
      S_Coil( #Event.%X14 )   // CYCLE RESET
   END_RUNG
   // the same network as SCL:
   #_w1 := #AlwaysTrue AND #"PHT Selected";
   #_w2 := #_w1 AND (#Status = 2);
   #_w3 := #_w2 AND NOT #Re3;   // rising edge
   #Re3 := #_w2;
   IF #_w3 THEN
       #Event.%X8 := TRUE;   // PRESSURIZE STARTED
   END_IF;
   #_w4 := #_w1 AND (#Status = 3);
   #_w5 := #_w4 AND NOT #Re4;   // rising edge
   #Re4 := #_w4;
   IF #_w5 THEN
       #Event.%X9 := TRUE;   // STABILIZE STARTED
   END_IF;
   #_w6 := #_w1 AND (#Status = 4);
   #_w7 := #_w6 AND NOT #Re5;   // rising edge
   #Re5 := #_w6;
   IF #_w7 THEN
       #Event.%X10 := TRUE;   // PRESSURE HOLD STARTED
   END_IF;
   #_w8 := #_w1 AND #Abort AND NOT #Re13;   // rising edge of #Abort
   #Re13 := #Abort;
   #_w9 := #_w1 AND #HoldTimer.DONE_BIT AND NOT #Re14;   // rising edge of #HoldTimer.DONE_BIT
   #Re14 := #HoldTimer.DONE_BIT;
   #_w10 := (#_w1 AND (#Status = 5) AND NOT #HoldTimer.DONE_BIT) OR #_w8 OR #_w9;
   #_w11 := #_w10 AND NOT #Re12;   // rising edge
   #Re12 := #_w10;
   IF #_w11 THEN
       #Event.%X11 := TRUE;   // PRESSURE RELEASE STARTED
   END_IF;
   #_w12 := #_w1 AND #HoldTimer.TIME_START AND NOT #Re15;   // rising edge of #HoldTimer.TIME_START
   #Re15 := #HoldTimer.TIME_START;
   IF #_w12 AND NOT "AlwaysTRUE" THEN
       #Event.%X1 := TRUE;   // FOR HOLD TIME
   END_IF;
   #_w13 := #_w1 AND #Stop AND NOT #Re7;   // rising edge of #Stop
   #Re7 := #Stop;
   IF #_w13 THEN
       #Event.%X13 := TRUE;   // CYCLE PAUSED
   END_IF;
   #_w14 := #_w1 AND #Popup2Enable AND #StartupMsg2 AND NOT #Re11;   // rising edge of #StartupMsg2
   #Re11 := #StartupMsg2;
   IF #_w14 THEN
       #Event.%X0 := TRUE;   // WAITING FOR ACK
   END_IF;
   #_w15 := #AlwaysTrue AND #CycleOver AND NOT #Re8;   // rising edge of #CycleOver
   #Re8 := #CycleOver;
   IF #_w15 AND NOT #ResetBit THEN
       #Event.%X12 := TRUE;   // PHT OVER
   END_IF;
   #_w16 := #AlwaysTrue AND #Abort AND NOT #Re10;   // rising edge of #Abort
   #Re10 := #Abort;
   IF #_w16 THEN
       #Event.%X14 := TRUE;   // CYCLE RESET
   END_IF;
END_REGION

REGION Network 29: End Message
   RUNG wire#powerrail
      Contact( #CycleOver )
      S_Coil( #EndMsg )
   END_RUNG
   RUNG wire#powerrail
      Contact( #EndMsgAck )
      wire#w1
      R_Coil( #EndMsg )
   END_RUNG
   RUNG wire#w1
      R_Coil( #CycleOver )
   END_RUNG
   // the same network as SCL:
   IF #CycleOver THEN #EndMsg := TRUE; END_IF;
   IF #EndMsgAck THEN
       #EndMsg := FALSE;
       #CycleOver := FALSE;
   END_IF;
END_REGION

REGION Network 30: Manual Abort
   RUNG wire#powerrail
      Contact( #Abort )
      S_Coil( #ResetBit )
   END_RUNG
   // the same network as SCL:
   IF #Abort THEN #ResetBit := TRUE; END_IF;
END_REGION

REGION Network 31: Reset
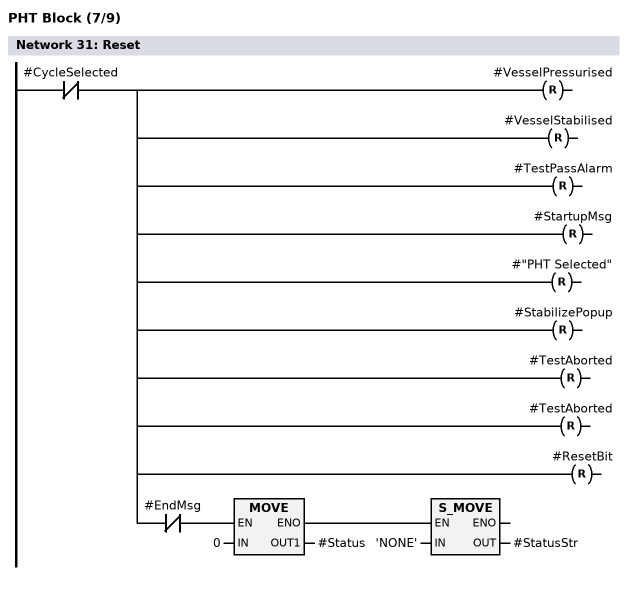
   RUNG wire#powerrail
      I_Contact( #CycleSelected )
      wire#w1
      R_Coil( #VesselPressurised )
   END_RUNG
   RUNG wire#w1
      R_Coil( #VesselStabilised )
   END_RUNG
   RUNG wire#w1
      R_Coil( #TestPassAlarm )
   END_RUNG
   RUNG wire#w1
      R_Coil( #StartupMsg )
   END_RUNG
   RUNG wire#w1
      R_Coil( #"PHT Selected" )
   END_RUNG
   RUNG wire#w1
      R_Coil( #StabilizePopup )
   END_RUNG
   RUNG wire#w1
      R_Coil( #TestAborted )
   END_RUNG
   RUNG wire#w1
      R_Coil( #TestAborted )
   END_RUNG
   RUNG wire#w1
      R_Coil( #ResetBit )
   END_RUNG
   RUNG wire#w1
      I_Contact( #EndMsg )
      { S7_GenerateENO := "TRUE" } Move(in := 0, out1 => #Status)
      S_Move(in := 'NONE', out => #StatusStr)
   END_RUNG
   // the same network as SCL:
   // ENO of a box is taken as its EN; it also drops when the box reports an error
   IF NOT #CycleSelected THEN
       #VesselPressurised := FALSE;
       #VesselStabilised := FALSE;
       #TestPassAlarm := FALSE;
       #StartupMsg := FALSE;
       #"PHT Selected" := FALSE;
       #StabilizePopup := FALSE;
       #TestAborted := FALSE;
       #TestAborted := FALSE;
       #ResetBit := FALSE;
   END_IF;
   IF NOT #CycleSelected AND NOT #EndMsg THEN
       #Status := 0;
       #StatusStr := 'NONE';
   END_IF;
END_REGION

REGION Network 32: Event reset
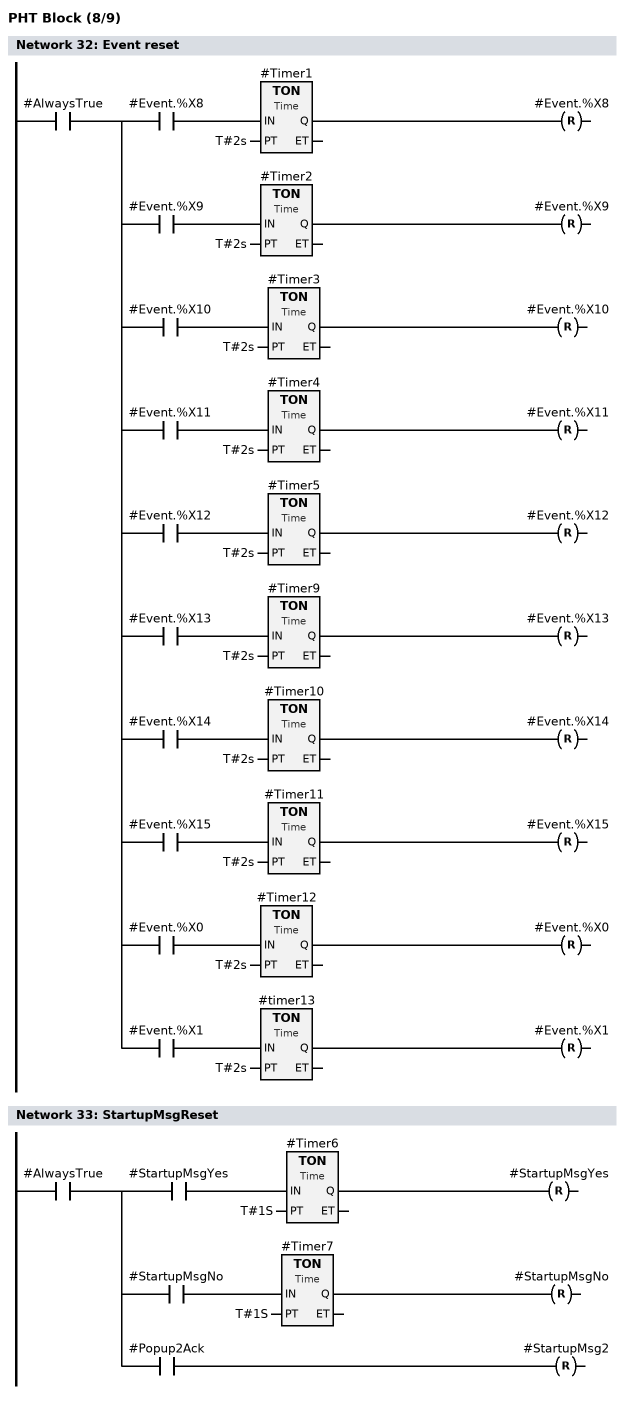
   RUNG wire#powerrail
      Contact( #AlwaysTrue )
      wire#w1
      Contact( #Event.%X8 )
      { S7_Templates := "time_type := Time" } #Timer1.TON(pt := T#2s, et =>)
      R_Coil( #Event.%X8 )
   END_RUNG
   RUNG wire#w1
      Contact( #Event.%X9 )
      { S7_Templates := "time_type := Time" } #Timer2.TON(pt := T#2s, et =>)
      R_Coil( #Event.%X9 )
   END_RUNG
   RUNG wire#w1
      Contact( #Event.%X10 )
      { S7_Templates := "time_type := Time" } #Timer3.TON(pt := T#2s, et =>)
      R_Coil( #Event.%X10 )
   END_RUNG
   RUNG wire#w1
      Contact( #Event.%X11 )
      { S7_Templates := "time_type := Time" } #Timer4.TON(pt := T#2s, et =>)
      R_Coil( #Event.%X11 )
   END_RUNG
   RUNG wire#w1
      Contact( #Event.%X12 )
      { S7_Templates := "time_type := Time" } #Timer5.TON(pt := T#2s, et =>)
      R_Coil( #Event.%X12 )
   END_RUNG
   RUNG wire#w1
      Contact( #Event.%X13 )
      { S7_Templates := "time_type := Time" } #Timer9.TON(pt := T#2s, et =>)
      R_Coil( #Event.%X13 )
   END_RUNG
   RUNG wire#w1
      Contact( #Event.%X14 )
      { S7_Templates := "time_type := Time" } #Timer10.TON(pt := T#2s, et =>)
      R_Coil( #Event.%X14 )
   END_RUNG
   RUNG wire#w1
      Contact( #Event.%X15 )
      { S7_Templates := "time_type := Time" } #Timer11.TON(pt := T#2s, et =>)
      R_Coil( #Event.%X15 )
   END_RUNG
   RUNG wire#w1
      Contact( #Event.%X0 )
      { S7_Templates := "time_type := Time" } #Timer12.TON(pt := T#2s, et =>)
      R_Coil( #Event.%X0 )
   END_RUNG
   RUNG wire#w1
      Contact( #Event.%X1 )
      { S7_Templates := "time_type := Time" } #timer13.TON(pt := T#2s, et =>)
      R_Coil( #Event.%X1 )
   END_RUNG
   // the same network as SCL:
   #Timer1(IN := #AlwaysTrue AND #Event.%X8, PT := T#2s);   // TON
   IF #Timer1.Q THEN #Event.%X8 := FALSE; END_IF;
   #Timer2(IN := #AlwaysTrue AND #Event.%X9, PT := T#2s);   // TON
   IF #Timer2.Q THEN #Event.%X9 := FALSE; END_IF;
   #Timer3(IN := #AlwaysTrue AND #Event.%X10, PT := T#2s);   // TON
   IF #Timer3.Q THEN #Event.%X10 := FALSE; END_IF;
   #Timer4(IN := #AlwaysTrue AND #Event.%X11, PT := T#2s);   // TON
   IF #Timer4.Q THEN #Event.%X11 := FALSE; END_IF;
   #Timer5(IN := #AlwaysTrue AND #Event.%X12, PT := T#2s);   // TON
   IF #Timer5.Q THEN #Event.%X12 := FALSE; END_IF;
   #Timer9(IN := #AlwaysTrue AND #Event.%X13, PT := T#2s);   // TON
   IF #Timer9.Q THEN #Event.%X13 := FALSE; END_IF;
   #Timer10(IN := #AlwaysTrue AND #Event.%X14, PT := T#2s);   // TON
   IF #Timer10.Q THEN #Event.%X14 := FALSE; END_IF;
   #Timer11(IN := #AlwaysTrue AND #Event.%X15, PT := T#2s);   // TON
   IF #Timer11.Q THEN #Event.%X15 := FALSE; END_IF;
   #Timer12(IN := #AlwaysTrue AND #Event.%X0, PT := T#2s);   // TON
   IF #Timer12.Q THEN #Event.%X0 := FALSE; END_IF;
   #timer13(IN := #AlwaysTrue AND #Event.%X1, PT := T#2s);   // TON
   IF #timer13.Q THEN #Event.%X1 := FALSE; END_IF;
END_REGION

REGION Network 33: StartupMsgReset
   RUNG wire#powerrail
      Contact( #AlwaysTrue )
      wire#w1
      Contact( #StartupMsgYes )
      { S7_Templates := "time_type := Time" } #Timer6.TON(pt := T#1S, et =>)
      R_Coil( #StartupMsgYes )
   END_RUNG
   RUNG wire#w1
      Contact( #StartupMsgNo )
      { S7_Templates := "time_type := Time" } #Timer7.TON(pt := T#1S, et =>)
      R_Coil( #StartupMsgNo )
   END_RUNG
   RUNG wire#w1
      Contact( #Popup2Ack )
      R_Coil( #StartupMsg2 )
   END_RUNG
   // the same network as SCL:
   #Timer6(IN := #AlwaysTrue AND #StartupMsgYes, PT := T#1S);   // TON
   IF #Timer6.Q THEN #StartupMsgYes := FALSE; END_IF;
   #Timer7(IN := #AlwaysTrue AND #StartupMsgNo, PT := T#1S);   // TON
   IF #Timer7.Q THEN #StartupMsgNo := FALSE; END_IF;
   IF #AlwaysTrue AND #Popup2Ack THEN #StartupMsg2 := FALSE; END_IF;
END_REGION

REGION Network 35: Line Print interval
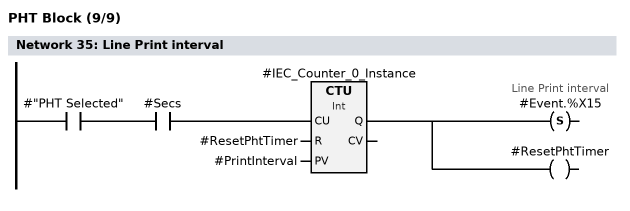
   RUNG wire#powerrail
      Contact( #"PHT Selected" )
      Contact( #Secs )
      { S7_Templates := "value_type := Int" } #IEC_Counter_0_Instance.CTU(r := #ResetPhtTimer, pv := #PrintInterval, cv =>)
      wire#w1
      S_Coil( #Event.%X15 )   // Line Print interval
   END_RUNG
   RUNG wire#w1
      Coil( #ResetPhtTimer )
   END_RUNG
   // the same network as SCL:
   #IEC_Counter_0_Instance(CU := #"PHT Selected" AND #Secs, R := #ResetPhtTimer, PV := #PrintInterval);   // CTU
   IF #IEC_Counter_0_Instance.Q THEN
       #Event.%X15 := TRUE;   // Line Print interval
   END_IF;
   #ResetPhtTimer := #IEC_Counter_0_Instance.Q;
END_REGION
END_FUNCTION_BLOCK
